// TIA Portal V20 export
FUNCTION "CallCycleTimerMapping" : Void   // FC4, LAD
// stored: SetENOAutomatically false
   VAR CONSTANT
      TRUE : Bool := TRUE;
   END_VAR
BEGIN

REGION Network 1: cycleTimerDataSet[1]
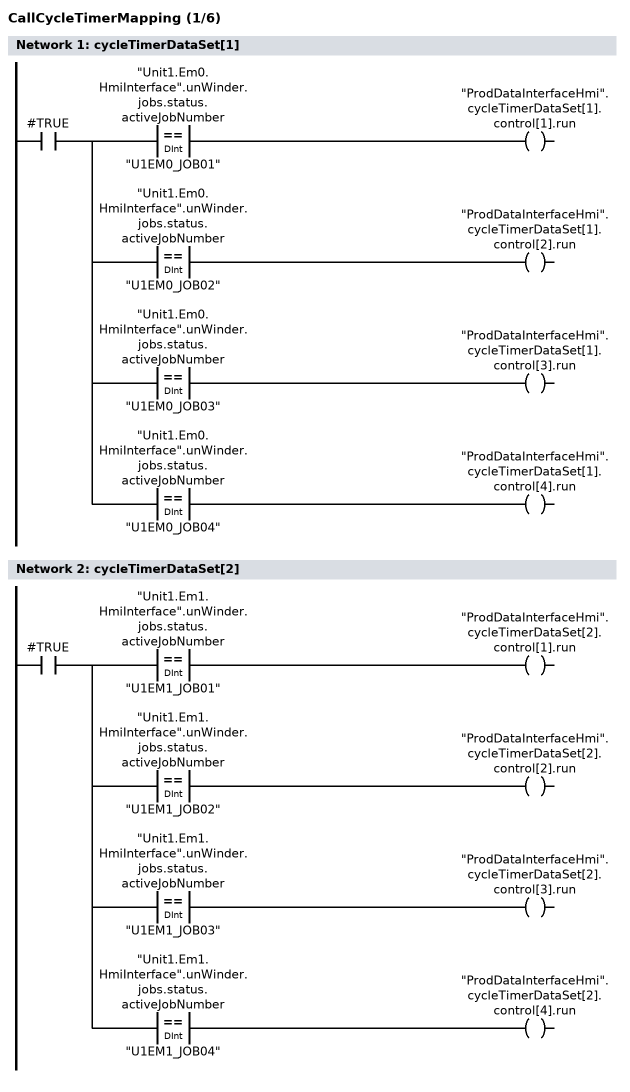
   RUNG wire#powerrail
      Contact( #TRUE )
      wire#w1
      { S7_Templates := "SrcType := DInt" } EQ_Contact(in1 := "Unit1.Em0.HmiInterface".unWinder.jobs.status.activeJobNumber, in2 := "U1EM0_JOB01")
      Coil( "ProdDataInterfaceHmi".cycleTimerDataSet[1].control[1].run )
   END_RUNG
   RUNG wire#w1
      { S7_Templates := "SrcType := DInt" } EQ_Contact(in1 := "Unit1.Em0.HmiInterface".unWinder.jobs.status.activeJobNumber, in2 := "U1EM0_JOB02")
      Coil( "ProdDataInterfaceHmi".cycleTimerDataSet[1].control[2].run )
   END_RUNG
   RUNG wire#w1
      { S7_Templates := "SrcType := DInt" } EQ_Contact(in1 := "Unit1.Em0.HmiInterface".unWinder.jobs.status.activeJobNumber, in2 := "U1EM0_JOB03")
      Coil( "ProdDataInterfaceHmi".cycleTimerDataSet[1].control[3].run )
   END_RUNG
   RUNG wire#w1
      { S7_Templates := "SrcType := DInt" } EQ_Contact(in1 := "Unit1.Em0.HmiInterface".unWinder.jobs.status.activeJobNumber, in2 := "U1EM0_JOB04")
      Coil( "ProdDataInterfaceHmi".cycleTimerDataSet[1].control[4].run )
   END_RUNG
   // the same network as SCL:
   "ProdDataInterfaceHmi".cycleTimerDataSet[1].control[1].run := #TRUE AND ("Unit1.Em0.HmiInterface".unWinder.jobs.status.activeJobNumber = "U1EM0_JOB01");
   "ProdDataInterfaceHmi".cycleTimerDataSet[1].control[2].run := #TRUE AND ("Unit1.Em0.HmiInterface".unWinder.jobs.status.activeJobNumber = "U1EM0_JOB02");
   "ProdDataInterfaceHmi".cycleTimerDataSet[1].control[3].run := #TRUE AND ("Unit1.Em0.HmiInterface".unWinder.jobs.status.activeJobNumber = "U1EM0_JOB03");
   "ProdDataInterfaceHmi".cycleTimerDataSet[1].control[4].run := #TRUE AND ("Unit1.Em0.HmiInterface".unWinder.jobs.status.activeJobNumber = "U1EM0_JOB04");
END_REGION

REGION Network 2: cycleTimerDataSet[2]
   RUNG wire#powerrail
      Contact( #TRUE )
      wire#w1
      { S7_Templates := "SrcType := DInt" } EQ_Contact(in1 := "Unit1.Em1.HmiInterface".unWinder.jobs.status.activeJobNumber, in2 := "U1EM1_JOB01")
      Coil( "ProdDataInterfaceHmi".cycleTimerDataSet[2].control[1].run )
   END_RUNG
   RUNG wire#w1
      { S7_Templates := "SrcType := DInt" } EQ_Contact(in1 := "Unit1.Em1.HmiInterface".unWinder.jobs.status.activeJobNumber, in2 := "U1EM1_JOB02")
      Coil( "ProdDataInterfaceHmi".cycleTimerDataSet[2].control[2].run )
   END_RUNG
   RUNG wire#w1
      { S7_Templates := "SrcType := DInt" } EQ_Contact(in1 := "Unit1.Em1.HmiInterface".unWinder.jobs.status.activeJobNumber, in2 := "U1EM1_JOB03")
      Coil( "ProdDataInterfaceHmi".cycleTimerDataSet[2].control[3].run )
   END_RUNG
   RUNG wire#w1
      { S7_Templates := "SrcType := DInt" } EQ_Contact(in1 := "Unit1.Em1.HmiInterface".unWinder.jobs.status.activeJobNumber, in2 := "U1EM1_JOB04")
      Coil( "ProdDataInterfaceHmi".cycleTimerDataSet[2].control[4].run )
   END_RUNG
   // the same network as SCL:
   "ProdDataInterfaceHmi".cycleTimerDataSet[2].control[1].run := #TRUE AND ("Unit1.Em1.HmiInterface".unWinder.jobs.status.activeJobNumber = "U1EM1_JOB01");
   "ProdDataInterfaceHmi".cycleTimerDataSet[2].control[2].run := #TRUE AND ("Unit1.Em1.HmiInterface".unWinder.jobs.status.activeJobNumber = "U1EM1_JOB02");
   "ProdDataInterfaceHmi".cycleTimerDataSet[2].control[3].run := #TRUE AND ("Unit1.Em1.HmiInterface".unWinder.jobs.status.activeJobNumber = "U1EM1_JOB03");
   "ProdDataInterfaceHmi".cycleTimerDataSet[2].control[4].run := #TRUE AND ("Unit1.Em1.HmiInterface".unWinder.jobs.status.activeJobNumber = "U1EM1_JOB04");
END_REGION

REGION Network 3: cycleTimerDataSet[3]
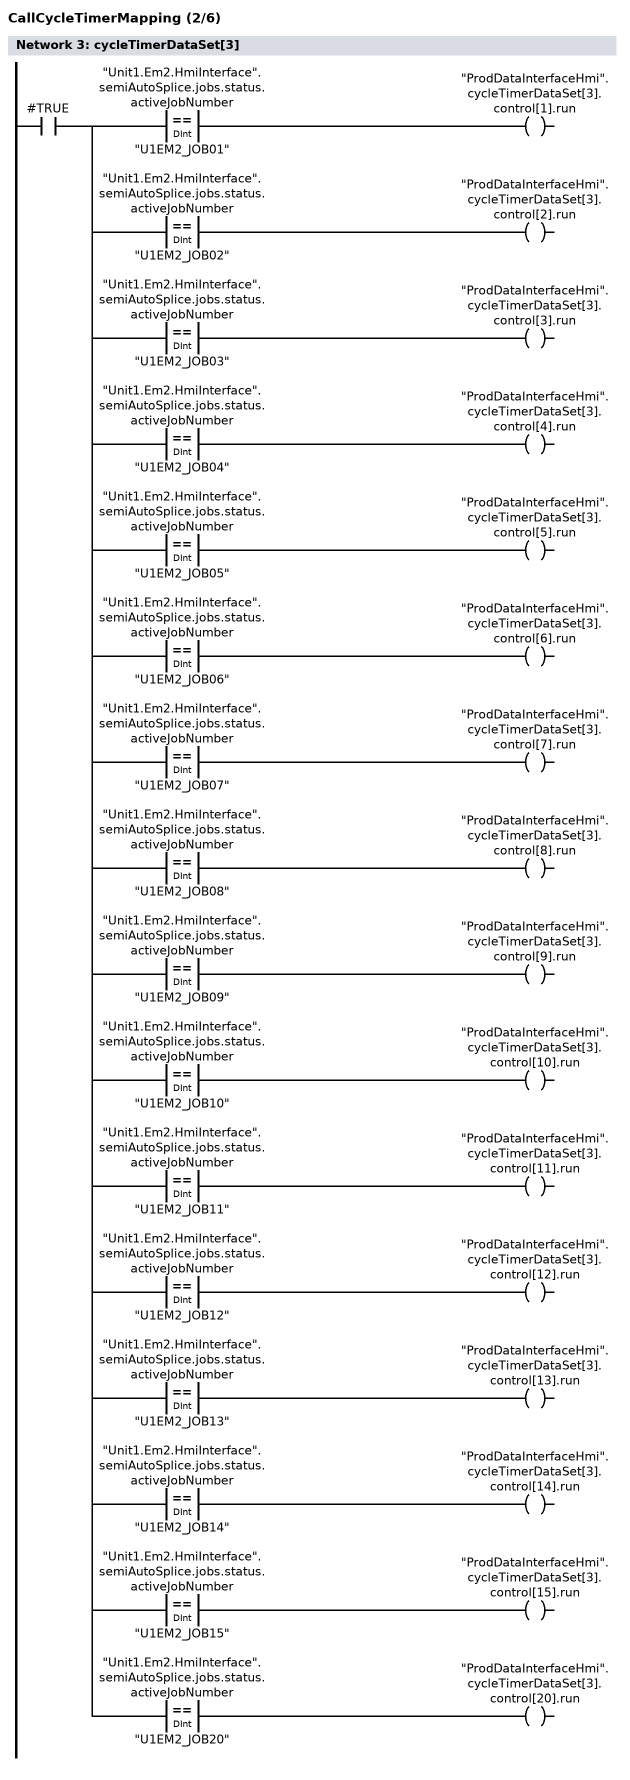
   RUNG wire#powerrail
      Contact( #TRUE )
      wire#w1
      { S7_Templates := "SrcType := DInt" } EQ_Contact(in1 := "Unit1.Em2.HmiInterface".semiAutoSplice.jobs.status.activeJobNumber, in2 := "U1EM2_JOB01")
      Coil( "ProdDataInterfaceHmi".cycleTimerDataSet[3].control[1].run )
   END_RUNG
   RUNG wire#w1
      { S7_Templates := "SrcType := DInt" } EQ_Contact(in1 := "Unit1.Em2.HmiInterface".semiAutoSplice.jobs.status.activeJobNumber, in2 := "U1EM2_JOB02")
      Coil( "ProdDataInterfaceHmi".cycleTimerDataSet[3].control[2].run )
   END_RUNG
   RUNG wire#w1
      { S7_Templates := "SrcType := DInt" } EQ_Contact(in1 := "Unit1.Em2.HmiInterface".semiAutoSplice.jobs.status.activeJobNumber, in2 := "U1EM2_JOB03")
      Coil( "ProdDataInterfaceHmi".cycleTimerDataSet[3].control[3].run )
   END_RUNG
   RUNG wire#w1
      { S7_Templates := "SrcType := DInt" } EQ_Contact(in1 := "Unit1.Em2.HmiInterface".semiAutoSplice.jobs.status.activeJobNumber, in2 := "U1EM2_JOB04")
      Coil( "ProdDataInterfaceHmi".cycleTimerDataSet[3].control[4].run )
   END_RUNG
   RUNG wire#w1
      { S7_Templates := "SrcType := DInt" } EQ_Contact(in1 := "Unit1.Em2.HmiInterface".semiAutoSplice.jobs.status.activeJobNumber, in2 := "U1EM2_JOB05")
      Coil( "ProdDataInterfaceHmi".cycleTimerDataSet[3].control[5].run )
   END_RUNG
   RUNG wire#w1
      { S7_Templates := "SrcType := DInt" } EQ_Contact(in1 := "Unit1.Em2.HmiInterface".semiAutoSplice.jobs.status.activeJobNumber, in2 := "U1EM2_JOB06")
      Coil( "ProdDataInterfaceHmi".cycleTimerDataSet[3].control[6].run )
   END_RUNG
   RUNG wire#w1
      { S7_Templates := "SrcType := DInt" } EQ_Contact(in1 := "Unit1.Em2.HmiInterface".semiAutoSplice.jobs.status.activeJobNumber, in2 := "U1EM2_JOB07")
      Coil( "ProdDataInterfaceHmi".cycleTimerDataSet[3].control[7].run )
   END_RUNG
   RUNG wire#w1
      { S7_Templates := "SrcType := DInt" } EQ_Contact(in1 := "Unit1.Em2.HmiInterface".semiAutoSplice.jobs.status.activeJobNumber, in2 := "U1EM2_JOB08")
      Coil( "ProdDataInterfaceHmi".cycleTimerDataSet[3].control[8].run )
   END_RUNG
   RUNG wire#w1
      { S7_Templates := "SrcType := DInt" } EQ_Contact(in1 := "Unit1.Em2.HmiInterface".semiAutoSplice.jobs.status.activeJobNumber, in2 := "U1EM2_JOB09")
      Coil( "ProdDataInterfaceHmi".cycleTimerDataSet[3].control[9].run )
   END_RUNG
   RUNG wire#w1
      { S7_Templates := "SrcType := DInt" } EQ_Contact(in1 := "Unit1.Em2.HmiInterface".semiAutoSplice.jobs.status.activeJobNumber, in2 := "U1EM2_JOB10")
      Coil( "ProdDataInterfaceHmi".cycleTimerDataSet[3].control[10].run )
   END_RUNG
   RUNG wire#w1
      { S7_Templates := "SrcType := DInt" } EQ_Contact(in1 := "Unit1.Em2.HmiInterface".semiAutoSplice.jobs.status.activeJobNumber, in2 := "U1EM2_JOB11")
      Coil( "ProdDataInterfaceHmi".cycleTimerDataSet[3].control[11].run )
   END_RUNG
   RUNG wire#w1
      { S7_Templates := "SrcType := DInt" } EQ_Contact(in1 := "Unit1.Em2.HmiInterface".semiAutoSplice.jobs.status.activeJobNumber, in2 := "U1EM2_JOB12")
      Coil( "ProdDataInterfaceHmi".cycleTimerDataSet[3].control[12].run )
   END_RUNG
   RUNG wire#w1
      { S7_Templates := "SrcType := DInt" } EQ_Contact(in1 := "Unit1.Em2.HmiInterface".semiAutoSplice.jobs.status.activeJobNumber, in2 := "U1EM2_JOB13")
      Coil( "ProdDataInterfaceHmi".cycleTimerDataSet[3].control[13].run )
   END_RUNG
   RUNG wire#w1
      { S7_Templates := "SrcType := DInt" } EQ_Contact(in1 := "Unit1.Em2.HmiInterface".semiAutoSplice.jobs.status.activeJobNumber, in2 := "U1EM2_JOB14")
      Coil( "ProdDataInterfaceHmi".cycleTimerDataSet[3].control[14].run )
   END_RUNG
   RUNG wire#w1
      { S7_Templates := "SrcType := DInt" } EQ_Contact(in1 := "Unit1.Em2.HmiInterface".semiAutoSplice.jobs.status.activeJobNumber, in2 := "U1EM2_JOB15")
      Coil( "ProdDataInterfaceHmi".cycleTimerDataSet[3].control[15].run )
   END_RUNG
   RUNG wire#w1
      { S7_Templates := "SrcType := DInt" } EQ_Contact(in1 := "Unit1.Em2.HmiInterface".semiAutoSplice.jobs.status.activeJobNumber, in2 := "U1EM2_JOB20")
      Coil( "ProdDataInterfaceHmi".cycleTimerDataSet[3].control[20].run )
   END_RUNG
   // the same network as SCL:
   "ProdDataInterfaceHmi".cycleTimerDataSet[3].control[1].run := #TRUE AND ("Unit1.Em2.HmiInterface".semiAutoSplice.jobs.status.activeJobNumber = "U1EM2_JOB01");
   "ProdDataInterfaceHmi".cycleTimerDataSet[3].control[2].run := #TRUE AND ("Unit1.Em2.HmiInterface".semiAutoSplice.jobs.status.activeJobNumber = "U1EM2_JOB02");
   "ProdDataInterfaceHmi".cycleTimerDataSet[3].control[3].run := #TRUE AND ("Unit1.Em2.HmiInterface".semiAutoSplice.jobs.status.activeJobNumber = "U1EM2_JOB03");
   "ProdDataInterfaceHmi".cycleTimerDataSet[3].control[4].run := #TRUE AND ("Unit1.Em2.HmiInterface".semiAutoSplice.jobs.status.activeJobNumber = "U1EM2_JOB04");
   "ProdDataInterfaceHmi".cycleTimerDataSet[3].control[5].run := #TRUE AND ("Unit1.Em2.HmiInterface".semiAutoSplice.jobs.status.activeJobNumber = "U1EM2_JOB05");
   "ProdDataInterfaceHmi".cycleTimerDataSet[3].control[6].run := #TRUE AND ("Unit1.Em2.HmiInterface".semiAutoSplice.jobs.status.activeJobNumber = "U1EM2_JOB06");
   "ProdDataInterfaceHmi".cycleTimerDataSet[3].control[7].run := #TRUE AND ("Unit1.Em2.HmiInterface".semiAutoSplice.jobs.status.activeJobNumber = "U1EM2_JOB07");
   "ProdDataInterfaceHmi".cycleTimerDataSet[3].control[8].run := #TRUE AND ("Unit1.Em2.HmiInterface".semiAutoSplice.jobs.status.activeJobNumber = "U1EM2_JOB08");
   "ProdDataInterfaceHmi".cycleTimerDataSet[3].control[9].run := #TRUE AND ("Unit1.Em2.HmiInterface".semiAutoSplice.jobs.status.activeJobNumber = "U1EM2_JOB09");
   "ProdDataInterfaceHmi".cycleTimerDataSet[3].control[10].run := #TRUE AND ("Unit1.Em2.HmiInterface".semiAutoSplice.jobs.status.activeJobNumber = "U1EM2_JOB10");
   "ProdDataInterfaceHmi".cycleTimerDataSet[3].control[11].run := #TRUE AND ("Unit1.Em2.HmiInterface".semiAutoSplice.jobs.status.activeJobNumber = "U1EM2_JOB11");
   "ProdDataInterfaceHmi".cycleTimerDataSet[3].control[12].run := #TRUE AND ("Unit1.Em2.HmiInterface".semiAutoSplice.jobs.status.activeJobNumber = "U1EM2_JOB12");
   "ProdDataInterfaceHmi".cycleTimerDataSet[3].control[13].run := #TRUE AND ("Unit1.Em2.HmiInterface".semiAutoSplice.jobs.status.activeJobNumber = "U1EM2_JOB13");
   "ProdDataInterfaceHmi".cycleTimerDataSet[3].control[14].run := #TRUE AND ("Unit1.Em2.HmiInterface".semiAutoSplice.jobs.status.activeJobNumber = "U1EM2_JOB14");
   "ProdDataInterfaceHmi".cycleTimerDataSet[3].control[15].run := #TRUE AND ("Unit1.Em2.HmiInterface".semiAutoSplice.jobs.status.activeJobNumber = "U1EM2_JOB15");
   "ProdDataInterfaceHmi".cycleTimerDataSet[3].control[20].run := #TRUE AND ("Unit1.Em2.HmiInterface".semiAutoSplice.jobs.status.activeJobNumber = "U1EM2_JOB20");
END_REGION

REGION Network 4: cycleTimerDataSet[4]
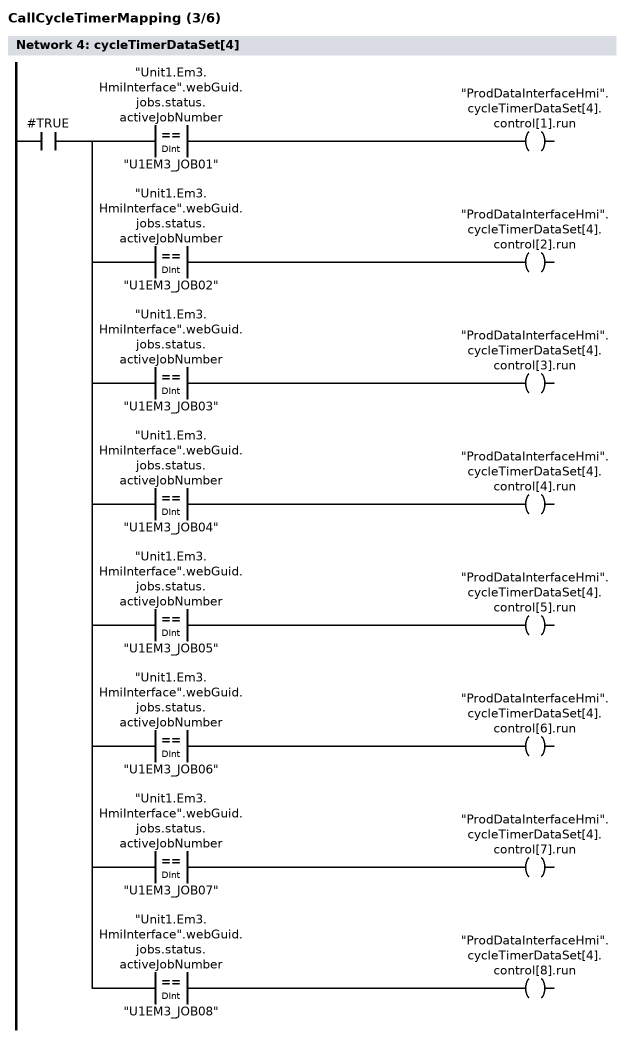
   RUNG wire#powerrail
      Contact( #TRUE )
      wire#w1
      { S7_Templates := "SrcType := DInt" } EQ_Contact(in1 := "Unit1.Em3.HmiInterface".webGuid.jobs.status.activeJobNumber, in2 := "U1EM3_JOB01")
      Coil( "ProdDataInterfaceHmi".cycleTimerDataSet[4].control[1].run )
   END_RUNG
   RUNG wire#w1
      { S7_Templates := "SrcType := DInt" } EQ_Contact(in1 := "Unit1.Em3.HmiInterface".webGuid.jobs.status.activeJobNumber, in2 := "U1EM3_JOB02")
      Coil( "ProdDataInterfaceHmi".cycleTimerDataSet[4].control[2].run )
   END_RUNG
   RUNG wire#w1
      { S7_Templates := "SrcType := DInt" } EQ_Contact(in1 := "Unit1.Em3.HmiInterface".webGuid.jobs.status.activeJobNumber, in2 := "U1EM3_JOB03")
      Coil( "ProdDataInterfaceHmi".cycleTimerDataSet[4].control[3].run )
   END_RUNG
   RUNG wire#w1
      { S7_Templates := "SrcType := DInt" } EQ_Contact(in1 := "Unit1.Em3.HmiInterface".webGuid.jobs.status.activeJobNumber, in2 := "U1EM3_JOB04")
      Coil( "ProdDataInterfaceHmi".cycleTimerDataSet[4].control[4].run )
   END_RUNG
   RUNG wire#w1
      { S7_Templates := "SrcType := DInt" } EQ_Contact(in1 := "Unit1.Em3.HmiInterface".webGuid.jobs.status.activeJobNumber, in2 := "U1EM3_JOB05")
      Coil( "ProdDataInterfaceHmi".cycleTimerDataSet[4].control[5].run )
   END_RUNG
   RUNG wire#w1
      { S7_Templates := "SrcType := DInt" } EQ_Contact(in1 := "Unit1.Em3.HmiInterface".webGuid.jobs.status.activeJobNumber, in2 := "U1EM3_JOB06")
      Coil( "ProdDataInterfaceHmi".cycleTimerDataSet[4].control[6].run )
   END_RUNG
   RUNG wire#w1
      { S7_Templates := "SrcType := DInt" } EQ_Contact(in1 := "Unit1.Em3.HmiInterface".webGuid.jobs.status.activeJobNumber, in2 := "U1EM3_JOB07")
      Coil( "ProdDataInterfaceHmi".cycleTimerDataSet[4].control[7].run )
   END_RUNG
   RUNG wire#w1
      { S7_Templates := "SrcType := DInt" } EQ_Contact(in1 := "Unit1.Em3.HmiInterface".webGuid.jobs.status.activeJobNumber, in2 := "U1EM3_JOB08")
      Coil( "ProdDataInterfaceHmi".cycleTimerDataSet[4].control[8].run )
   END_RUNG
   // the same network as SCL:
   "ProdDataInterfaceHmi".cycleTimerDataSet[4].control[1].run := #TRUE AND ("Unit1.Em3.HmiInterface".webGuid.jobs.status.activeJobNumber = "U1EM3_JOB01");
   "ProdDataInterfaceHmi".cycleTimerDataSet[4].control[2].run := #TRUE AND ("Unit1.Em3.HmiInterface".webGuid.jobs.status.activeJobNumber = "U1EM3_JOB02");
   "ProdDataInterfaceHmi".cycleTimerDataSet[4].control[3].run := #TRUE AND ("Unit1.Em3.HmiInterface".webGuid.jobs.status.activeJobNumber = "U1EM3_JOB03");
   "ProdDataInterfaceHmi".cycleTimerDataSet[4].control[4].run := #TRUE AND ("Unit1.Em3.HmiInterface".webGuid.jobs.status.activeJobNumber = "U1EM3_JOB04");
   "ProdDataInterfaceHmi".cycleTimerDataSet[4].control[5].run := #TRUE AND ("Unit1.Em3.HmiInterface".webGuid.jobs.status.activeJobNumber = "U1EM3_JOB05");
   "ProdDataInterfaceHmi".cycleTimerDataSet[4].control[6].run := #TRUE AND ("Unit1.Em3.HmiInterface".webGuid.jobs.status.activeJobNumber = "U1EM3_JOB06");
   "ProdDataInterfaceHmi".cycleTimerDataSet[4].control[7].run := #TRUE AND ("Unit1.Em3.HmiInterface".webGuid.jobs.status.activeJobNumber = "U1EM3_JOB07");
   "ProdDataInterfaceHmi".cycleTimerDataSet[4].control[8].run := #TRUE AND ("Unit1.Em3.HmiInterface".webGuid.jobs.status.activeJobNumber = "U1EM3_JOB08");
END_REGION

REGION Network 5: cycleTimerDataSet[5]
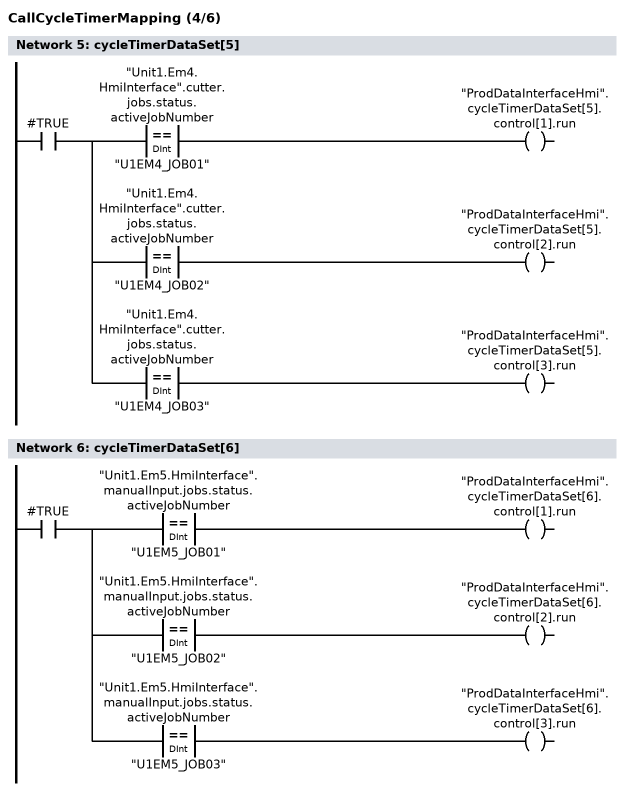
   RUNG wire#powerrail
      Contact( #TRUE )
      wire#w1
      { S7_Templates := "SrcType := DInt" } EQ_Contact(in1 := "Unit1.Em4.HmiInterface".cutter.jobs.status.activeJobNumber, in2 := "U1EM4_JOB01")
      Coil( "ProdDataInterfaceHmi".cycleTimerDataSet[5].control[1].run )
   END_RUNG
   RUNG wire#w1
      { S7_Templates := "SrcType := DInt" } EQ_Contact(in1 := "Unit1.Em4.HmiInterface".cutter.jobs.status.activeJobNumber, in2 := "U1EM4_JOB02")
      Coil( "ProdDataInterfaceHmi".cycleTimerDataSet[5].control[2].run )
   END_RUNG
   RUNG wire#w1
      { S7_Templates := "SrcType := DInt" } EQ_Contact(in1 := "Unit1.Em4.HmiInterface".cutter.jobs.status.activeJobNumber, in2 := "U1EM4_JOB03")
      Coil( "ProdDataInterfaceHmi".cycleTimerDataSet[5].control[3].run )
   END_RUNG
   // the same network as SCL:
   "ProdDataInterfaceHmi".cycleTimerDataSet[5].control[1].run := #TRUE AND ("Unit1.Em4.HmiInterface".cutter.jobs.status.activeJobNumber = "U1EM4_JOB01");
   "ProdDataInterfaceHmi".cycleTimerDataSet[5].control[2].run := #TRUE AND ("Unit1.Em4.HmiInterface".cutter.jobs.status.activeJobNumber = "U1EM4_JOB02");
   "ProdDataInterfaceHmi".cycleTimerDataSet[5].control[3].run := #TRUE AND ("Unit1.Em4.HmiInterface".cutter.jobs.status.activeJobNumber = "U1EM4_JOB03");
END_REGION

REGION Network 6: cycleTimerDataSet[6]
   RUNG wire#powerrail
      Contact( #TRUE )
      wire#w1
      { S7_Templates := "SrcType := DInt" } EQ_Contact(in1 := "Unit1.Em5.HmiInterface".manualInput.jobs.status.activeJobNumber, in2 := "U1EM5_JOB01")
      Coil( "ProdDataInterfaceHmi".cycleTimerDataSet[6].control[1].run )
   END_RUNG
   RUNG wire#w1
      { S7_Templates := "SrcType := DInt" } EQ_Contact(in1 := "Unit1.Em5.HmiInterface".manualInput.jobs.status.activeJobNumber, in2 := "U1EM5_JOB02")
      Coil( "ProdDataInterfaceHmi".cycleTimerDataSet[6].control[2].run )
   END_RUNG
   RUNG wire#w1
      { S7_Templates := "SrcType := DInt" } EQ_Contact(in1 := "Unit1.Em5.HmiInterface".manualInput.jobs.status.activeJobNumber, in2 := "U1EM5_JOB03")
      Coil( "ProdDataInterfaceHmi".cycleTimerDataSet[6].control[3].run )
   END_RUNG
   // the same network as SCL:
   "ProdDataInterfaceHmi".cycleTimerDataSet[6].control[1].run := #TRUE AND ("Unit1.Em5.HmiInterface".manualInput.jobs.status.activeJobNumber = "U1EM5_JOB01");
   "ProdDataInterfaceHmi".cycleTimerDataSet[6].control[2].run := #TRUE AND ("Unit1.Em5.HmiInterface".manualInput.jobs.status.activeJobNumber = "U1EM5_JOB02");
   "ProdDataInterfaceHmi".cycleTimerDataSet[6].control[3].run := #TRUE AND ("Unit1.Em5.HmiInterface".manualInput.jobs.status.activeJobNumber = "U1EM5_JOB03");
END_REGION

REGION Network 7: cycleTimerDataSet[7]
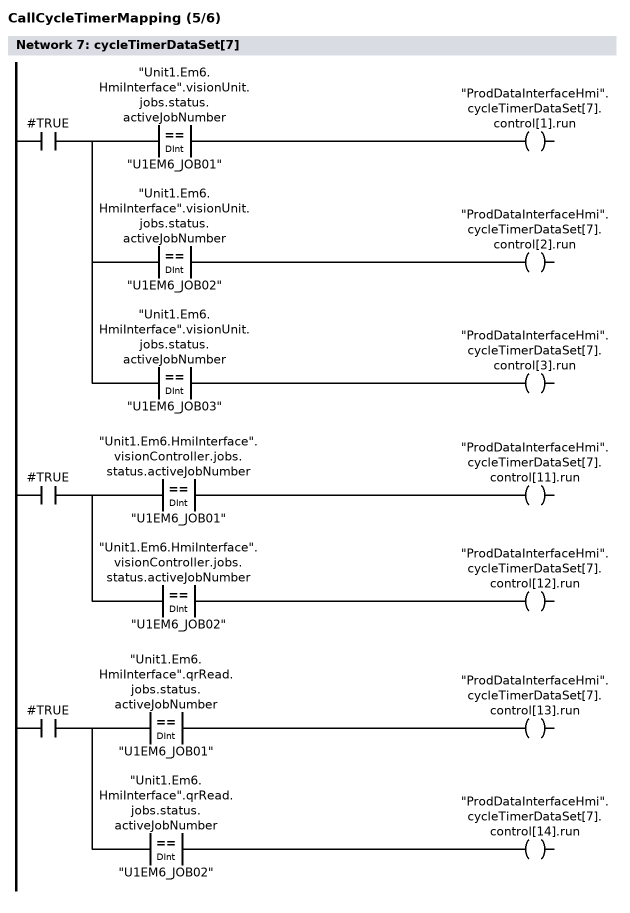
   RUNG wire#powerrail
      Contact( #TRUE )
      wire#w1
      { S7_Templates := "SrcType := DInt" } EQ_Contact(in1 := "Unit1.Em6.HmiInterface".visionUnit.jobs.status.activeJobNumber, in2 := "U1EM6_JOB01")
      Coil( "ProdDataInterfaceHmi".cycleTimerDataSet[7].control[1].run )
   END_RUNG
   RUNG wire#w1
      { S7_Templates := "SrcType := DInt" } EQ_Contact(in1 := "Unit1.Em6.HmiInterface".visionUnit.jobs.status.activeJobNumber, in2 := "U1EM6_JOB02")
      Coil( "ProdDataInterfaceHmi".cycleTimerDataSet[7].control[2].run )
   END_RUNG
   RUNG wire#w1
      { S7_Templates := "SrcType := DInt" } EQ_Contact(in1 := "Unit1.Em6.HmiInterface".visionUnit.jobs.status.activeJobNumber, in2 := "U1EM6_JOB03")
      Coil( "ProdDataInterfaceHmi".cycleTimerDataSet[7].control[3].run )
   END_RUNG
   RUNG wire#powerrail
      Contact( #TRUE )
      wire#w2
      { S7_Templates := "SrcType := DInt" } EQ_Contact(in1 := "Unit1.Em6.HmiInterface".visionController.jobs.status.activeJobNumber, in2 := "U1EM6_JOB01")
      Coil( "ProdDataInterfaceHmi".cycleTimerDataSet[7].control[11].run )
   END_RUNG
   RUNG wire#w2
      { S7_Templates := "SrcType := DInt" } EQ_Contact(in1 := "Unit1.Em6.HmiInterface".visionController.jobs.status.activeJobNumber, in2 := "U1EM6_JOB02")
      Coil( "ProdDataInterfaceHmi".cycleTimerDataSet[7].control[12].run )
   END_RUNG
   RUNG wire#powerrail
      Contact( #TRUE )
      wire#w3
      { S7_Templates := "SrcType := DInt" } EQ_Contact(in1 := "Unit1.Em6.HmiInterface".qrRead.jobs.status.activeJobNumber, in2 := "U1EM6_JOB01")
      Coil( "ProdDataInterfaceHmi".cycleTimerDataSet[7].control[13].run )
   END_RUNG
   RUNG wire#w3
      { S7_Templates := "SrcType := DInt" } EQ_Contact(in1 := "Unit1.Em6.HmiInterface".qrRead.jobs.status.activeJobNumber, in2 := "U1EM6_JOB02")
      Coil( "ProdDataInterfaceHmi".cycleTimerDataSet[7].control[14].run )
   END_RUNG
   // the same network as SCL:
   "ProdDataInterfaceHmi".cycleTimerDataSet[7].control[1].run := #TRUE AND ("Unit1.Em6.HmiInterface".visionUnit.jobs.status.activeJobNumber = "U1EM6_JOB01");
   "ProdDataInterfaceHmi".cycleTimerDataSet[7].control[2].run := #TRUE AND ("Unit1.Em6.HmiInterface".visionUnit.jobs.status.activeJobNumber = "U1EM6_JOB02");
   "ProdDataInterfaceHmi".cycleTimerDataSet[7].control[3].run := #TRUE AND ("Unit1.Em6.HmiInterface".visionUnit.jobs.status.activeJobNumber = "U1EM6_JOB03");
   "ProdDataInterfaceHmi".cycleTimerDataSet[7].control[11].run := #TRUE AND ("Unit1.Em6.HmiInterface".visionController.jobs.status.activeJobNumber = "U1EM6_JOB01");
   "ProdDataInterfaceHmi".cycleTimerDataSet[7].control[12].run := #TRUE AND ("Unit1.Em6.HmiInterface".visionController.jobs.status.activeJobNumber = "U1EM6_JOB02");
   "ProdDataInterfaceHmi".cycleTimerDataSet[7].control[13].run := #TRUE AND ("Unit1.Em6.HmiInterface".qrRead.jobs.status.activeJobNumber = "U1EM6_JOB01");
   "ProdDataInterfaceHmi".cycleTimerDataSet[7].control[14].run := #TRUE AND ("Unit1.Em6.HmiInterface".qrRead.jobs.status.activeJobNumber = "U1EM6_JOB02");
END_REGION

REGION Network 8: cycleTimerDataSet[8]
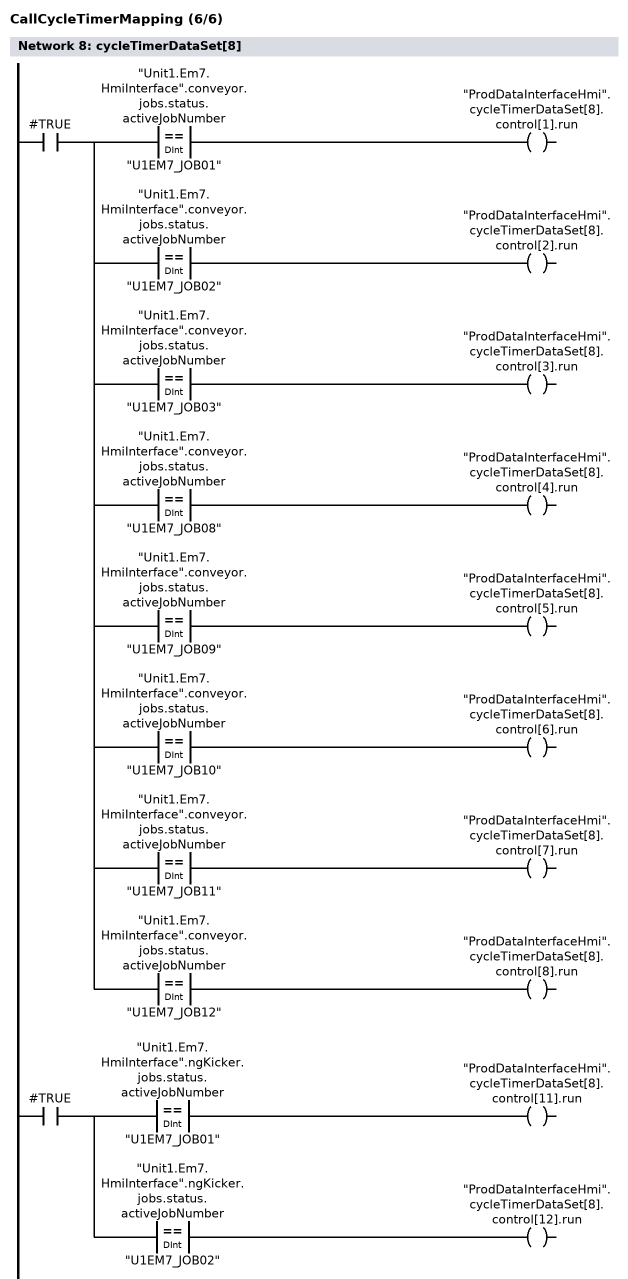
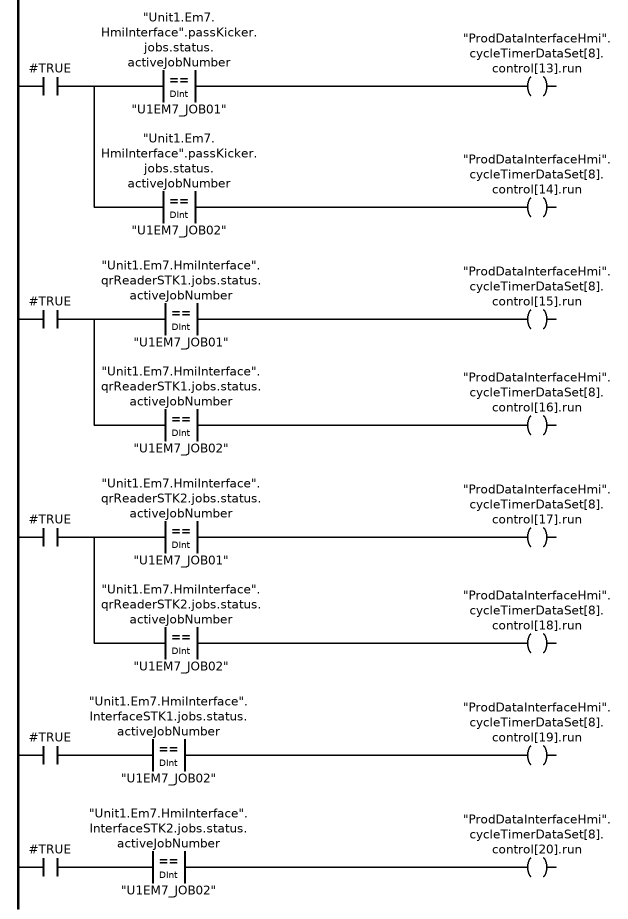
   RUNG wire#powerrail
      Contact( #TRUE )
      wire#w1
      { S7_Templates := "SrcType := DInt" } EQ_Contact(in1 := "Unit1.Em7.HmiInterface".conveyor.jobs.status.activeJobNumber, in2 := "U1EM7_JOB01")
      Coil( "ProdDataInterfaceHmi".cycleTimerDataSet[8].control[1].run )
   END_RUNG
   RUNG wire#w1
      { S7_Templates := "SrcType := DInt" } EQ_Contact(in1 := "Unit1.Em7.HmiInterface".conveyor.jobs.status.activeJobNumber, in2 := "U1EM7_JOB02")
      Coil( "ProdDataInterfaceHmi".cycleTimerDataSet[8].control[2].run )
   END_RUNG
   RUNG wire#w1
      { S7_Templates := "SrcType := DInt" } EQ_Contact(in1 := "Unit1.Em7.HmiInterface".conveyor.jobs.status.activeJobNumber, in2 := "U1EM7_JOB03")
      Coil( "ProdDataInterfaceHmi".cycleTimerDataSet[8].control[3].run )
   END_RUNG
   RUNG wire#w1
      { S7_Templates := "SrcType := DInt" } EQ_Contact(in1 := "Unit1.Em7.HmiInterface".conveyor.jobs.status.activeJobNumber, in2 := "U1EM7_JOB08")
      Coil( "ProdDataInterfaceHmi".cycleTimerDataSet[8].control[4].run )
   END_RUNG
   RUNG wire#w1
      { S7_Templates := "SrcType := DInt" } EQ_Contact(in1 := "Unit1.Em7.HmiInterface".conveyor.jobs.status.activeJobNumber, in2 := "U1EM7_JOB09")
      Coil( "ProdDataInterfaceHmi".cycleTimerDataSet[8].control[5].run )
   END_RUNG
   RUNG wire#w1
      { S7_Templates := "SrcType := DInt" } EQ_Contact(in1 := "Unit1.Em7.HmiInterface".conveyor.jobs.status.activeJobNumber, in2 := "U1EM7_JOB10")
      Coil( "ProdDataInterfaceHmi".cycleTimerDataSet[8].control[6].run )
   END_RUNG
   RUNG wire#w1
      { S7_Templates := "SrcType := DInt" } EQ_Contact(in1 := "Unit1.Em7.HmiInterface".conveyor.jobs.status.activeJobNumber, in2 := "U1EM7_JOB11")
      Coil( "ProdDataInterfaceHmi".cycleTimerDataSet[8].control[7].run )
   END_RUNG
   RUNG wire#w1
      { S7_Templates := "SrcType := DInt" } EQ_Contact(in1 := "Unit1.Em7.HmiInterface".conveyor.jobs.status.activeJobNumber, in2 := "U1EM7_JOB12")
      Coil( "ProdDataInterfaceHmi".cycleTimerDataSet[8].control[8].run )
   END_RUNG
   RUNG wire#powerrail
      Contact( #TRUE )
      wire#w2
      { S7_Templates := "SrcType := DInt" } EQ_Contact(in1 := "Unit1.Em7.HmiInterface".ngKicker.jobs.status.activeJobNumber, in2 := "U1EM7_JOB01")
      Coil( "ProdDataInterfaceHmi".cycleTimerDataSet[8].control[11].run )
   END_RUNG
   RUNG wire#w2
      { S7_Templates := "SrcType := DInt" } EQ_Contact(in1 := "Unit1.Em7.HmiInterface".ngKicker.jobs.status.activeJobNumber, in2 := "U1EM7_JOB02")
      Coil( "ProdDataInterfaceHmi".cycleTimerDataSet[8].control[12].run )
   END_RUNG
   RUNG wire#powerrail
      Contact( #TRUE )
      wire#w3
      { S7_Templates := "SrcType := DInt" } EQ_Contact(in1 := "Unit1.Em7.HmiInterface".passKicker.jobs.status.activeJobNumber, in2 := "U1EM7_JOB01")
      Coil( "ProdDataInterfaceHmi".cycleTimerDataSet[8].control[13].run )
   END_RUNG
   RUNG wire#w3
      { S7_Templates := "SrcType := DInt" } EQ_Contact(in1 := "Unit1.Em7.HmiInterface".passKicker.jobs.status.activeJobNumber, in2 := "U1EM7_JOB02")
      Coil( "ProdDataInterfaceHmi".cycleTimerDataSet[8].control[14].run )
   END_RUNG
   RUNG wire#powerrail
      Contact( #TRUE )
      wire#w4
      { S7_Templates := "SrcType := DInt" } EQ_Contact(in1 := "Unit1.Em7.HmiInterface".qrReaderSTK1.jobs.status.activeJobNumber, in2 := "U1EM7_JOB01")
      Coil( "ProdDataInterfaceHmi".cycleTimerDataSet[8].control[15].run )
   END_RUNG
   RUNG wire#w4
      { S7_Templates := "SrcType := DInt" } EQ_Contact(in1 := "Unit1.Em7.HmiInterface".qrReaderSTK1.jobs.status.activeJobNumber, in2 := "U1EM7_JOB02")
      Coil( "ProdDataInterfaceHmi".cycleTimerDataSet[8].control[16].run )
   END_RUNG
   RUNG wire#powerrail
      Contact( #TRUE )
      wire#w5
      { S7_Templates := "SrcType := DInt" } EQ_Contact(in1 := "Unit1.Em7.HmiInterface".qrReaderSTK2.jobs.status.activeJobNumber, in2 := "U1EM7_JOB01")
      Coil( "ProdDataInterfaceHmi".cycleTimerDataSet[8].control[17].run )
   END_RUNG
   RUNG wire#w5
      { S7_Templates := "SrcType := DInt" } EQ_Contact(in1 := "Unit1.Em7.HmiInterface".qrReaderSTK2.jobs.status.activeJobNumber, in2 := "U1EM7_JOB02")
      Coil( "ProdDataInterfaceHmi".cycleTimerDataSet[8].control[18].run )
   END_RUNG
   RUNG wire#powerrail
      Contact( #TRUE )
      { S7_Templates := "SrcType := DInt" } EQ_Contact(in1 := "Unit1.Em7.HmiInterface".InterfaceSTK1.jobs.status.activeJobNumber, in2 := "U1EM7_JOB02")
      Coil( "ProdDataInterfaceHmi".cycleTimerDataSet[8].control[19].run )
   END_RUNG
   RUNG wire#powerrail
      Contact( #TRUE )
      { S7_Templates := "SrcType := DInt" } EQ_Contact(in1 := "Unit1.Em7.HmiInterface".InterfaceSTK2.jobs.status.activeJobNumber, in2 := "U1EM7_JOB02")
      Coil( "ProdDataInterfaceHmi".cycleTimerDataSet[8].control[20].run )
   END_RUNG
   // the same network as SCL:
   "ProdDataInterfaceHmi".cycleTimerDataSet[8].control[1].run := #TRUE AND ("Unit1.Em7.HmiInterface".conveyor.jobs.status.activeJobNumber = "U1EM7_JOB01");
   "ProdDataInterfaceHmi".cycleTimerDataSet[8].control[2].run := #TRUE AND ("Unit1.Em7.HmiInterface".conveyor.jobs.status.activeJobNumber = "U1EM7_JOB02");
   "ProdDataInterfaceHmi".cycleTimerDataSet[8].control[3].run := #TRUE AND ("Unit1.Em7.HmiInterface".conveyor.jobs.status.activeJobNumber = "U1EM7_JOB03");
   "ProdDataInterfaceHmi".cycleTimerDataSet[8].control[4].run := #TRUE AND ("Unit1.Em7.HmiInterface".conveyor.jobs.status.activeJobNumber = "U1EM7_JOB08");
   "ProdDataInterfaceHmi".cycleTimerDataSet[8].control[5].run := #TRUE AND ("Unit1.Em7.HmiInterface".conveyor.jobs.status.activeJobNumber = "U1EM7_JOB09");
   "ProdDataInterfaceHmi".cycleTimerDataSet[8].control[6].run := #TRUE AND ("Unit1.Em7.HmiInterface".conveyor.jobs.status.activeJobNumber = "U1EM7_JOB10");
   "ProdDataInterfaceHmi".cycleTimerDataSet[8].control[7].run := #TRUE AND ("Unit1.Em7.HmiInterface".conveyor.jobs.status.activeJobNumber = "U1EM7_JOB11");
   "ProdDataInterfaceHmi".cycleTimerDataSet[8].control[8].run := #TRUE AND ("Unit1.Em7.HmiInterface".conveyor.jobs.status.activeJobNumber = "U1EM7_JOB12");
   "ProdDataInterfaceHmi".cycleTimerDataSet[8].control[11].run := #TRUE AND ("Unit1.Em7.HmiInterface".ngKicker.jobs.status.activeJobNumber = "U1EM7_JOB01");
   "ProdDataInterfaceHmi".cycleTimerDataSet[8].control[12].run := #TRUE AND ("Unit1.Em7.HmiInterface".ngKicker.jobs.status.activeJobNumber = "U1EM7_JOB02");
   "ProdDataInterfaceHmi".cycleTimerDataSet[8].control[13].run := #TRUE AND ("Unit1.Em7.HmiInterface".passKicker.jobs.status.activeJobNumber = "U1EM7_JOB01");
   "ProdDataInterfaceHmi".cycleTimerDataSet[8].control[14].run := #TRUE AND ("Unit1.Em7.HmiInterface".passKicker.jobs.status.activeJobNumber = "U1EM7_JOB02");
   "ProdDataInterfaceHmi".cycleTimerDataSet[8].control[15].run := #TRUE AND ("Unit1.Em7.HmiInterface".qrReaderSTK1.jobs.status.activeJobNumber = "U1EM7_JOB01");
   "ProdDataInterfaceHmi".cycleTimerDataSet[8].control[16].run := #TRUE AND ("Unit1.Em7.HmiInterface".qrReaderSTK1.jobs.status.activeJobNumber = "U1EM7_JOB02");
   "ProdDataInterfaceHmi".cycleTimerDataSet[8].control[17].run := #TRUE AND ("Unit1.Em7.HmiInterface".qrReaderSTK2.jobs.status.activeJobNumber = "U1EM7_JOB01");
   "ProdDataInterfaceHmi".cycleTimerDataSet[8].control[18].run := #TRUE AND ("Unit1.Em7.HmiInterface".qrReaderSTK2.jobs.status.activeJobNumber = "U1EM7_JOB02");
   "ProdDataInterfaceHmi".cycleTimerDataSet[8].control[19].run := #TRUE AND ("Unit1.Em7.HmiInterface".InterfaceSTK1.jobs.status.activeJobNumber = "U1EM7_JOB02");
   "ProdDataInterfaceHmi".cycleTimerDataSet[8].control[20].run := #TRUE AND ("Unit1.Em7.HmiInterface".InterfaceSTK2.jobs.status.activeJobNumber = "U1EM7_JOB02");
END_REGION
END_FUNCTION
